// TIA Portal V20 export
DATA_BLOCK "InterfaceSignals"   // DB232
// stored: Access Published, InstanceOfName LER_SignalsInterface, InstanceOfType UDT
"LER_SignalsInterface"
   // VAR
   //    HMI_Select_Mode : Bool := FALSE;
   //    ButtonValue : Array[0..16] of "LER_SignalsInput";
   // END_VAR
BEGIN
   ButtonValue[0].ButtonLeft[0..15] := FALSE;
   ButtonValue[1].ButtonLeft[0..15] := FALSE;
   ButtonValue[2].ButtonLeft[0..15] := FALSE;
   ButtonValue[3].ButtonLeft[0..15] := FALSE;
   ButtonValue[4].ButtonLeft[0..15] := FALSE;
   ButtonValue[5].ButtonLeft[0..15] := FALSE;
   ButtonValue[6].ButtonLeft[0..15] := FALSE;
   ButtonValue[7].ButtonLeft[0..15] := FALSE;
   ButtonValue[8].ButtonLeft[0..15] := FALSE;
   ButtonValue[9].ButtonLeft[0..15] := FALSE;
   ButtonValue[10].ButtonLeft[0..15] := FALSE;
   ButtonValue[11].ButtonLeft[0..15] := FALSE;
   ButtonValue[12].ButtonLeft[0..15] := FALSE;
   ButtonValue[13].ButtonLeft[0..15] := FALSE;
   ButtonValue[14].ButtonLeft[0..15] := FALSE;
   ButtonValue[15].ButtonLeft[0..15] := FALSE;
   ButtonValue[16].ButtonLeft[0..15] := FALSE;
   ButtonValue[0].ButtonRight[0..15] := FALSE;
   ButtonValue[1].ButtonRight[0..15] := FALSE;
   ButtonValue[2].ButtonRight[0..15] := FALSE;
   ButtonValue[3].ButtonRight[0..15] := FALSE;
   ButtonValue[4].ButtonRight[0..15] := FALSE;
   ButtonValue[5].ButtonRight[0..15] := FALSE;
   ButtonValue[6].ButtonRight[0..15] := FALSE;
   ButtonValue[7].ButtonRight[0..15] := FALSE;
   ButtonValue[8].ButtonRight[0..15] := FALSE;
   ButtonValue[9].ButtonRight[0..15] := FALSE;
   ButtonValue[10].ButtonRight[0..15] := FALSE;
   ButtonValue[11].ButtonRight[0..15] := FALSE;
   ButtonValue[12].ButtonRight[0..15] := FALSE;
   ButtonValue[13].ButtonRight[0..15] := FALSE;
   ButtonValue[14].ButtonRight[0..15] := FALSE;
   ButtonValue[15].ButtonRight[0..15] := FALSE;
   ButtonValue[16].ButtonRight[0..15] := FALSE;
END_DATA_BLOCK
